PROGRAM MAIN
VAR
END_VAR

END_PROGRAM

(* stored: Version 1.1.0.1
   POU MAIN: Id {1546441b-9baa-4f37-9fcb-3e061acccb80} *)
